PROGRAM MAIN
VAR
	fbFoo1	:	MyNamespace01.FB_Foo;
	fbFoo2	:	MyNamespace02.FB_Foo;
	fbFoo3	:	FB_Foo;
END_VAR

fbFoo1();
fbFoo2();
fbFoo3();

END_PROGRAM

(* stored: Version 1.1.0.1, ProductVersion 3.1.4020.6
   POU MAIN: Id {b180a901-9060-4304-b58a-988ceafe4550}, SpecialFunc None *)
